{attribute 'linkalways'}
{attribute 'no_explicit_call' := 'This FB is a CLASS and must be accessed using methods or properties'}
{attribute 'enable_dynamic_creation'}
FUNCTION_BLOCK Node_F_VN_ConvertCartesianToPolarImagesExp EXTENDS VisionNode
VAR
    ipSrcImageX : _ITcVnImage;
    ipSrcImageY : _ITcVnImage;
    ipDestImageMag : _ITcVnImage;
    ipDestImageAng : _ITcVnImage;
    bAngleInDegrees : _BOOL(FALSE);
    hrPrev : _HRESULT(S_OK);
    hresult : _HRESULT(S_OK);
END_VAR

METHOD PUBLIC Clone : I_Node
VAR
    pNode : POINTER TO Node_F_VN_ConvertCartesianToPolarImagesExp;
END_VAR
pNode := __NEW(Node_F_VN_ConvertCartesianToPolarImagesExp);
Clone := pNode^;
END_METHOD

METHOD FB_init : BOOL
VAR_INPUT
    bInitRetains : BOOL;
    bInCopyCode : BOOL;
END_VAR
AddInput('ipSrcImageX', ipSrcImageX);
AddInput('ipSrcImageY', ipSrcImageY);
AddOutput('ipDestImageMag', ipDestImageMag);
AddOutput('ipDestImageAng', ipDestImageAng);
AddParameter('bAngleInDegrees', bAngleInDegrees);
AddInput('hrPrev', hrPrev);
AddOutput('hresult', hresult);
END_METHOD

METHOD PROTECTED OnExecute
hresult.Value := F_VN_ConvertCartesianToPolarImagesExp(
    ipSrcImageX := ipSrcImageX.Value,
    ipSrcImageY := ipSrcImageY.Value,
    ipDestImageMag := ipDestImageMag.Value,
    ipDestImageAng := ipDestImageAng.Value,
    bAngleInDegrees := bAngleInDegrees.Value,
    hrPrev := hrPrev.Value);
END_METHOD

METHOD PUBLIC PreExecutionCheck
VAR_INPUT
    Check : I_PreExecutionChecks;
END_VAR
Check.IsTrue(ipSrcImageX.IsValid, 'ipSrcImageX must contain an image');
Check.IsTrue(ipSrcImageX.IsElementType(ETcVnElementType.TCVN_ET_REAL) OR
             ipSrcImageX.IsElementType(ETcVnElementType.TCVN_ET_LREAL), 'Coordinate images must contain REAL or LREAL elements');
Check.IsTrue(ipSrcImageY.IsValid, 'ipSrcImageY must contain an image');
Check.IsTrue(ImagesHaveMatchingPixelFormats(ipSrcImageX.Value, ipSrcImageY.Value), 'Source images must have matching pixel formats');
Check.IsTrue(IsImage1SizeEqualToImage2Size(ipSrcImageX.Value, ipSrcImageY.Value), 'Source images must have matching dimensions');
END_METHOD

END_FUNCTION_BLOCK

(* stored: Version 1.1.0.1, ProductVersion 3.1.4026.19
   POU Node_F_VN_ConvertCartesianToPolarImagesExp: Id {2abfdd84-2ebe-41f9-93f2-7844acdf9eff}, SpecialFunc None
   Folder Constructor: Id {33fd06f6-30fd-4d9a-b7d6-f0e2ae8c0b90}
   Method Clone: Id {f3092413-1f30-41da-b38b-05da1519cea2}
   Method FB_init: Id {0cb4e752-9648-409c-9ba2-dd2e28c24e5b}
   Method OnExecute: Id {c7df21f7-3b4c-4bdf-bffd-7a4df64eda78}
   Method PreExecutionCheck: Id {1e724b13-ceff-451a-84b0-9bfbf5889953} *)
